% RSLogix 500 project PROC1_BLOWER_HOA_CONTROL_BAK000.RSS, saved by version 8.30.00.16 %
PROJECT "PROC1"    % processor: Bul.1763 MicroLogix 1100 Series B %

PROGRAM FILES
  LAD 2 "MAIN"  3 rungs
  LAD 3 "DIGITAL IO"  5 rungs
  LAD 4 "CONTROLS"  5 rungs

DATA FILES
  O0 OUTPUT  5 elements
  I1 INPUT  7 elements
  S2 STATUS  66 elements
  B3 BINARY  1 elements
  T4 TIMER  1 elements
  C5 COUNTER  1 elements
  R6 CONTROL  1 elements
  N7 INTEGER  1 elements
  F8 FLOAT  1 elements

LADDER 2 "MAIN"
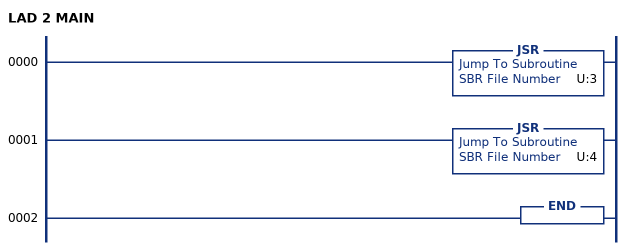
% Rung: 0 %
SOR JSR U:3 EOR
% Rung: 1 %
SOR JSR U:4 EOR
% Rung: 2 %
SOR END EOR

LADDER 3 "DIGITAL IO"
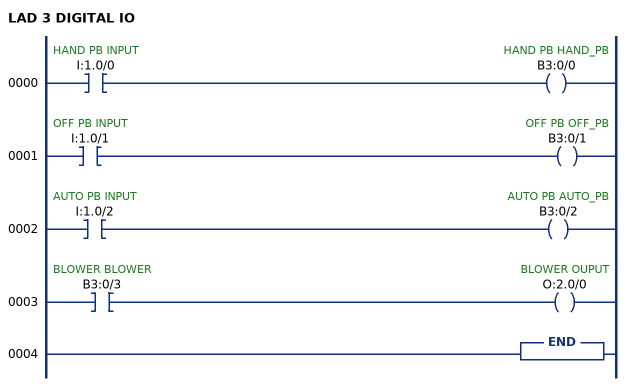
% Rung: 0 %
SOR XIC I:1.0/0 OTE B3:0/0 EOR
%   I:1.0/0  "HAND PB INPUT" %
%   B3:0/0  HAND_PB  "HAND PB" %
% Rung: 1 %
SOR XIC I:1.0/1 OTE B3:0/1 EOR
%   I:1.0/1  "OFF PB INPUT" %
%   B3:0/1  OFF_PB  "OFF PB" %
% Rung: 2 %
SOR XIC I:1.0/2 OTE B3:0/2 EOR
%   I:1.0/2  "AUTO PB INPUT" %
%   B3:0/2  AUTO_PB  "AUTO PB" %
% Rung: 3 %
SOR XIC B3:0/3 OTE O:2.0/0 EOR
%   B3:0/3  BLOWER  "BLOWER" %
%   O:2.0/0  "BLOWER OUPUT" %
% Rung: 4 %
SOR END EOR

LADDER 4 "CONTROLS"
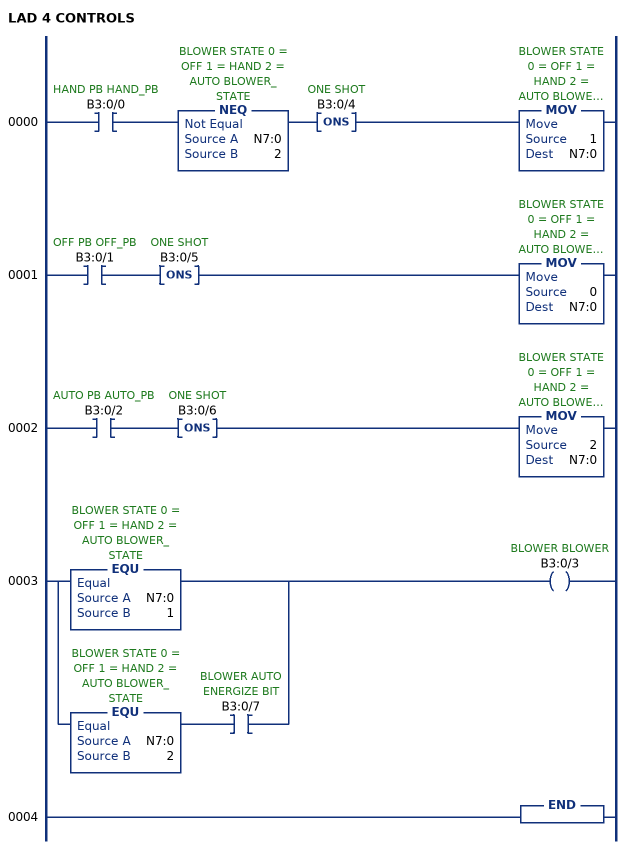
% Rung: 0 %
SOR XIC B3:0/0 NEQ N7:0 2 ONS B3:0/4 MOV 1 N7:0 EOR
%   B3:0/0  HAND_PB  "HAND PB" %
%   N7:0  BLOWER_STATE  "BLOWER STATE 0 = OFF 1 = HAND 2 = AUTO" %
%   B3:0/4  "ONE SHOT" %
% Rung: 1 %
SOR XIC B3:0/1 ONS B3:0/5 MOV 0 N7:0 EOR
%   B3:0/1  OFF_PB  "OFF PB" %
%   B3:0/5  "ONE SHOT" %
%   N7:0  BLOWER_STATE  "BLOWER STATE 0 = OFF 1 = HAND 2 = AUTO" %
% Rung: 2 %
SOR XIC B3:0/2 ONS B3:0/6 MOV 2 N7:0 EOR
%   B3:0/2  AUTO_PB  "AUTO PB" %
%   B3:0/6  "ONE SHOT" %
%   N7:0  BLOWER_STATE  "BLOWER STATE 0 = OFF 1 = HAND 2 = AUTO" %
% Rung: 3 %
SOR BST EQU N7:0 1 NXB EQU N7:0 2 XIC B3:0/7 BND OTE B3:0/3 EOR
%   N7:0  BLOWER_STATE  "BLOWER STATE 0 = OFF 1 = HAND 2 = AUTO" %
%   B3:0/7  "BLOWER AUTO ENERGIZE BIT" %
%   B3:0/3  BLOWER  "BLOWER" %
% Rung: 4 %
SOR END EOR
